VAR_GLOBAL CONSTANT
	PLCPRJ_BUFFER_SIZE					: UDINT := 1000;(* Max. internal fifo/receiver buffer size *)

	(* Some project specific error codes *)
	PLCPRJ_ERROR_SENDFIFO_OVERFLOW		: UDINT := 16#8103;
	PLCPRJ_ERROR_RECFIFO_OVERFLOW		: UDINT := 16#8104;
END_VAR

(* stored: Version 1.1.0.1, ProductVersion 3.1.0.20
   GVL Global_Variables: Id {6b661f4d-6075-4cd9-a960-2736d213cf6d} *)
